FUNCTION_BLOCK getSDODatenMotor
VAR_INPUT
	nSlaveAddr: UINT;
	nIndex: WORD;
END_VAR

VAR_OUTPUT
	// Ausglesene SDOs aus 9020 bzw. 9030
	Spannung: UINT;
	Strom: INT;
	Strombegrenzung: UINT;
	Regelfehler: INT;
	Geschwindigkeit: INT;
	Overloadtime: UINT;
	Overtemperature: BOOL;
	Torqueoverload: BOOL;
	Shortcircuit: BOOL;
END_VAR
	
VAR
	MotorspannungBlock: FB_EcCoESdoRead;	
	MotorstromBlock: FB_EcCoESdoRead;
	StrombegrenzungBlock: FB_EcCoESdoRead;
	RegelfehlerBlock: FB_EcCoESdoRead;
	GeschwindigkeitBlock: FB_EcCoESdoRead;
	OverloadTimeBlock: FB_EcCoESdoRead;
	Short_CircuitBlock: FB_EcCoESdoRead;
	Torque_OverloadBlock: FB_EcCoESdoRead;
	Over_TemperatureBlock: FB_EcCoESdoRead;

	trigger: BOOL;
	triggerStromSpannung: BOOL;
	TON_0: TON;
	TON_1: TON;
	TON_2: TON;
	TON_3: TON;
	ms: TIME;

END_VAR

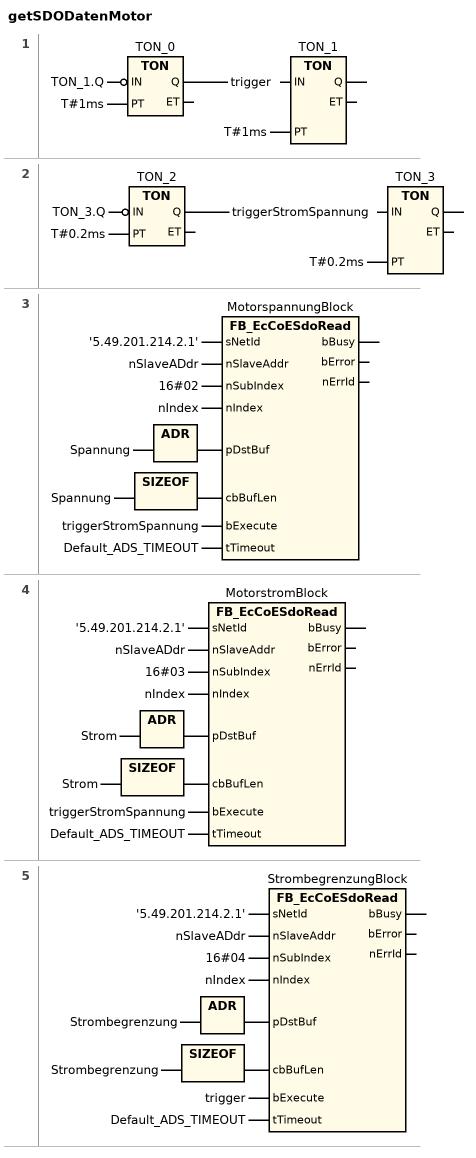
// NETWORK 1
TON_0(IN := NOT TON_1.Q, PT := T#1ms); // TON
trigger := TON_0.Q;
TON_1(IN := TON_0.Q, PT := T#1ms); // TON

// NETWORK 2
TON_2(IN := NOT TON_3.Q, PT := T#0.2ms); // TON
triggerStromSpannung := TON_2.Q;
TON_3(IN := TON_2.Q, PT := T#0.2ms); // TON

// NETWORK 3
MotorspannungBlock(
    sNetId := '5.49.201.214.2.1',
    nSlaveAddr := nSlaveADdr,
    nSubIndex := 16#02,
    nIndex := nIndex,
    pDstBuf := ADR(Spannung),
    cbBufLen := SIZEOF(Spannung),
    bExecute := triggerStromSpannung,
    tTimeout := Default_ADS_TIMEOUT); // FB_EcCoESdoRead

// NETWORK 4
MotorstromBlock(
    sNetId := '5.49.201.214.2.1',
    nSlaveAddr := nSlaveADdr,
    nSubIndex := 16#03,
    nIndex := nIndex,
    pDstBuf := ADR(Strom),
    cbBufLen := SIZEOF(Strom),
    bExecute := triggerStromSpannung,
    tTimeout := Default_ADS_TIMEOUT); // FB_EcCoESdoRead

// NETWORK 5
StrombegrenzungBlock(
    sNetId := '5.49.201.214.2.1',
    nSlaveAddr := nSlaveADdr,
    nSubIndex := 16#04,
    nIndex := nIndex,
    pDstBuf := ADR(Strombegrenzung),
    cbBufLen := SIZEOF(Strombegrenzung),
    bExecute := trigger,
    tTimeout := Default_ADS_TIMEOUT); // FB_EcCoESdoRead

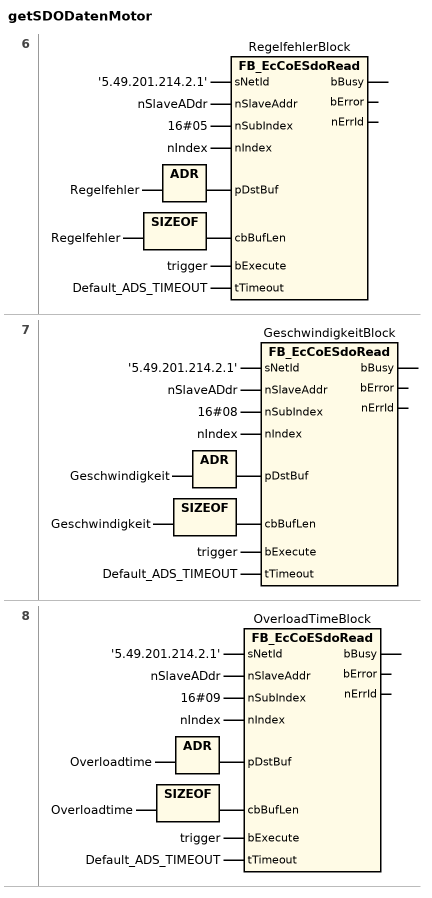
// NETWORK 6
RegelfehlerBlock(
    sNetId := '5.49.201.214.2.1',
    nSlaveAddr := nSlaveADdr,
    nSubIndex := 16#05,
    nIndex := nIndex,
    pDstBuf := ADR(Regelfehler),
    cbBufLen := SIZEOF(Regelfehler),
    bExecute := trigger,
    tTimeout := Default_ADS_TIMEOUT); // FB_EcCoESdoRead

// NETWORK 7
GeschwindigkeitBlock(
    sNetId := '5.49.201.214.2.1',
    nSlaveAddr := nSlaveADdr,
    nSubIndex := 16#08,
    nIndex := nIndex,
    pDstBuf := ADR(Geschwindigkeit),
    cbBufLen := SIZEOF(Geschwindigkeit),
    bExecute := trigger,
    tTimeout := Default_ADS_TIMEOUT); // FB_EcCoESdoRead

// NETWORK 8
OverloadTimeBlock(
    sNetId := '5.49.201.214.2.1',
    nSlaveAddr := nSlaveADdr,
    nSubIndex := 16#09,
    nIndex := nIndex,
    pDstBuf := ADR(Overloadtime),
    cbBufLen := SIZEOF(Overloadtime),
    bExecute := trigger,
    tTimeout := Default_ADS_TIMEOUT); // FB_EcCoESdoRead

END_FUNCTION_BLOCK

(* stored: Version 1.1.0.1, ProductVersion 3.1.4022.3
   POU getSDODatenMotor: Id {58be8c72-c68f-42e0-a6d5-ea46e21dd455}, SpecialFunc None *)
